    sTemp := 'IF(state,1,0))';

    StrConcatA(
        ADR(sTemp),
        ADR(sSQL),
        TO_INT(SIZEOF(sSQL))
    );


    // =================================================
    // WHERE
    // =================================================

    sTemp := ' FROM logs WHERE id BETWEEN ';

    StrConcatA(
        ADR(sTemp),
        ADR(sSQL),
        TO_INT(SIZEOF(sSQL))
    );

    sTemp := DWORD_TO_STRING(dwStartId);

    StrConcatA(
        ADR(sTemp),
        ADR(sSQL),
        TO_INT(SIZEOF(sSQL))
    );

    sTemp := ' AND ';

    StrConcatA(
        ADR(sTemp),
        ADR(sSQL),
        TO_INT(SIZEOF(sSQL))
    );


	sTemp := UDINT_TO_STRING(TO_UDINT(dwStartId) + TO_UDINT(uiCount));
	 
    StrConcatA(
        ADR(sTemp),
        ADR(sSQL),
        TO_INT(SIZEOF(sSQL))
    );

    // =================================================
    // ORDER
    // =================================================

    sTemp := ' ORDER BY id DESC;';

    StrConcatA(
        ADR(sTemp),
        ADR(sSQL),
        TO_INT(SIZEOF(sSQL))
    );

   

    // =================================================
    // MARIADB COMMAND
    // =================================================

    sCommand := '';

    sTemp :=
        'mariadb --socket=/var/lib/mysql/mysql.sock ';

    StrConcatA(
        ADR(sTemp),
        ADR(sCommand),
        TO_INT(SIZEOF(sCommand))
    );


    sTemp :=
        '-u root -pCTA-MariaDb1981! ';

    StrConcatA(
        ADR(sTemp),
        ADR(sCommand),
        TO_INT(SIZEOF(sCommand))
    );


    sTemp :=
        '--default-character-set=utf8mb4 CtaMariaDb ';

    StrConcatA(
        ADR(sTemp),
        ADR(sCommand),
        TO_INT(SIZEOF(sCommand))
    );


    sTemp :=
        '-N -B -e "';

    StrConcatA(
        ADR(sTemp),
        ADR(sCommand),
        TO_INT(SIZEOF(sCommand))
    );


    // SQL anhängen

    StrConcatA(
        ADR(sSQL),
        ADR(sCommand),
        TO_INT(SIZEOF(sCommand))
    );


    sTemp := '"';

    StrConcatA(
        ADR(sTemp),
        ADR(sCommand),
        TO_INT(SIZEOF(sCommand))
    );


    // =================================================
    // SQL AUSFÜHREN
    // =================================================

    sStdOut := '';

    diStdOutLen :=
        SysProcess_Implementation.SysProcessExecuteCommand2(
            pszCommand := sCommand,
            pszStdOut := sStdOut,
            udiStdOutLen := SIZEOF(sStdOut),
            pResult := ADR(Result)
        );


    // =================================================
    // FEHLER
    // =================================================

    IF Result <> CmpErrors.Errors.ERR_OK THEN

        xError := TRUE;
        xDone := FALSE;
        dwResult := 2;

    ELSE

        // =============================================
        // ERGEBNIS PARSEN
        // =============================================

        sRemaining := sStdOut;

        uiRead := 0;


        FOR i := 0 TO 13 DO

            IF uiRead >= uiCount THEN
                EXIT;
            END_IF;


            // -----------------------------------------
            // nächste Zeile suchen
            // MARIADB -B liefert LF
            // -----------------------------------------

            iPos := StrFindA(ADR(sRemaining), ADR(cLF),0);


            IF iPos > 0 THEN

                StrMidA(ADR(sRemaining),SIZEOF(sRemaining),iPos - 1,1,ADR(sRow),SIZEOF(sRow));

                StrDeleteA(ADR(sRemaining),  iPos,1);

            ELSE

                // letzte Zeile

                sRow := sRemaining;
                sRemaining := '';

            END_IF;


            // -----------------------------------------
            // leere Zeile ignorieren
            // -----------------------------------------

            IF LEN(sRow) > 0 THEN


                // =====================================
                // FELD 1 - ID
                // =====================================

                iPos := FIND(sRow, '\t');

                IF iPos > 0 THEN

                    sField := LEFT(sRow, iPos - 1);

                    StrDeleteA(ADR(sRow),iPos + 1,1);

                    aLogs[uiRead].id := TO_ULINT(sField);

                END_IF;


                // =====================================
                // FELD 2 - CREATED AT
                // =====================================

                iPos := FIND(sRow, '\t');

                IF iPos > 0 THEN

                    sField := LEFT(sRow, iPos - 1);

					StrDeleteA(ADR(sRow),iPos + 1,1);

                    IF LEN(sField) > 0 THEN
						sField := REPLACE(sField,'-',1,FIND(sField,' '));
                        aLogs[uiRead].createdAt := TO_DT(CONCAT('DT#',sField));
                    END_IF;

                END_IF;


                // =====================================
                // FELD 3 - EVENT TYPE
                // =====================================

                iPos := FIND(sRow, '\t');

                IF iPos > 0 THEN

                    sField := LEFT(sRow, iPos - 1);

					StrDeleteA(ADR(sRow),iPos + 1,1);

                    IF sField = 'ERROR' THEN
                        aLogs[uiRead].reportType :=
                            enReportType.Error;

                    ELSIF sField = 'WARNING' THEN
                        aLogs[uiRead].reportType :=
                            enReportType.Warning;

                    ELSIF sField = 'INFO' THEN
                        aLogs[uiRead].reportType :=
                            enReportType.Info;

                    ELSE
                        aLogs[uiRead].reportType :=
                            enReportType.Info;
                    END_IF;

                END_IF;


                // =====================================
                // FELD 4 - EVENT ID
                // =====================================

                iPos := FIND(sRow, '\t');

                IF iPos > 0 THEN

                    sField := LEFT(sRow, iPos - 1);

					StrDeleteA(ADR(sRow),iPos + 1,1);

                    aLogs[uiRead].reportId :=
                        TO_ULINT(sField);

                END_IF;


                // =====================================
                // FELD 5 - OBJECT NAME
                // =====================================

                iPos := FIND(sRow, '\t');

                IF iPos > 0 THEN

                    aLogs[uiRead].reporterText :=
                        LEFT(sRow, iPos - 1);

					StrDeleteA(ADR(sRow),iPos + 1,1);

                END_IF;


                // =====================================
                // FELD 6 - REPORT TEXT
                // =====================================

                iPos := FIND(sRow, '\t');

                IF iPos > 0 THEN

                    aLogs[uiRead].reportText :=
                        LEFT(sRow, iPos - 1);

					StrDeleteA(ADR(sRow),iPos + 1,1);

                END_IF;


                // =====================================
                // FELD 7 - DT FROM
                // =====================================

                iPos := FIND(sRow, '\t');

                IF iPos > 0 THEN

                    sField := LEFT(sRow, iPos - 1);

					StrDeleteA(ADR(sRow),iPos + 1,1);

                    IF LEN(sField) > 0 THEN
						sField := REPLACE(sField,'-',1,FIND(sField,' '));
                        aLogs[uiRead].dtFrom := TO_DT(CONCAT('DT#',sField));
                    END_IF;

                END_IF;


                // =====================================
                // FELD 8 - DT TO
                // =====================================

                iPos := FIND(sRow, '\t');

                IF iPos > 0 THEN

                    sField := LEFT(sRow, iPos - 1);

					StrDeleteA(ADR(sRow),iPos + 1,1);

                    IF LEN(sField) > 0 THEN
						sField := REPLACE(sField,'-',1,FIND(sField,' '));
                        aLogs[uiRead].dtTo := TO_DT(CONCAT('DT#',sField));
                    END_IF;

                END_IF;


                // =====================================
                // FELD 9 - IS QUITT
                // =====================================

                iPos := FIND(sRow, '\t');

                IF iPos > 0 THEN

                    sField := LEFT(sRow, iPos - 1);

					StrDeleteA(ADR(sRow),iPos + 1,1);

                    aLogs[uiRead].isQuitt := TO_BOOL(TO_INT(sField));

                END_IF;


                // =====================================
                // FELD 10 - REPORT TEXT LIST
                // =====================================

                iPos := FIND(sRow, '\t');

                IF iPos > 0 THEN

                    aLogs[uiRead].reportTextList :=
                        LEFT(sRow, iPos - 1);

					StrDeleteA(ADR(sRow),iPos + 1,1);

                END_IF;


                // =====================================
                // FELD 11 - TEXT ID
                // =====================================

                iPos := FIND(sRow, '\t');

                IF iPos > 0 THEN

                    sField := LEFT(sRow, iPos - 1);

					StrDeleteA(ADR(sRow),iPos + 1,1);

                    aLogs[uiRead].reportTextId :=
                        sField;

                END_IF;


                // =====================================
                // FELD 12 - ACKNOWLEDGEMENT
                // =====================================

                iPos := FIND(sRow, '\t');

                IF iPos > 0 THEN

                    sField := LEFT(sRow, iPos - 1);

					StrDeleteA(ADR(sRow),iPos + 1,1);

                    aLogs[uiRead].reportAcknowledgType :=
                        TO_USINT(sField);

                END_IF;


                // =====================================
                // FELD 13 - OBJECT ID
                // =====================================

                iPos := FIND(sRow, '\t');

                IF iPos > 0 THEN

                    aLogs[uiRead].objectId :=
                        LEFT(sRow, iPos - 1);

					StrDeleteA(ADR(sRow),iPos + 1,1);

                END_IF;


                // =====================================
                // FELD 14 - INSTANCE PATH
                // =====================================

                iPos := FIND(sRow, '\t');

                IF iPos > 0 THEN

                    aLogs[uiRead].instancePath :=
                        LEFT(sRow, iPos - 1);

					StrDeleteA(ADR(sRow),iPos + 1,1);

                END_IF;


                // =====================================
                // FELD 15 - ADDITIONAL TEXT
                // =====================================

                iPos := FIND(sRow, '\t');

                IF iPos > 0 THEN

                    aLogs[uiRead].additionalText :=
                        LEFT(sRow, iPos - 1);

					StrDeleteA(ADR(sRow),iPos + 1,1);

                END_IF;


                // =====================================
                // FELD 16 - PRIO
                // =====================================

                iPos := FIND(sRow, '\t');

                IF iPos > 0 THEN

                    sField := LEFT(sRow, iPos - 1);

					StrDeleteA(ADR(sRow),iPos + 1,1);

                    aLogs[uiRead].prio :=
                        TO_USINT(sField);

                END_IF;


                // =====================================
                // FELD 17 - IN STATE
                // =====================================

                iPos := FIND(sRow, '\t');

                IF iPos > 0 THEN

                    sField := LEFT(sRow, iPos - 1);

					StrDeleteA(ADR(sRow),iPos + 1,1);

                    aLogs[uiRead].reportIn := TO_BOOL(TO_INT(sField));
                END_IF;


                // =====================================
                // FELD 18 - STATE
                // =====================================

                IF LEN(sRow) > 0 THEN

                    aLogs[uiRead].stateActive := TO_BOOL(TO_INT(sRow));

                END_IF;


                // =====================================
                // DATENSATZ GÜLTIG
                // =====================================

                IF aLogs[uiRead].id > 0 THEN

                    uiRead := uiRead + 1;

                END_IF;

            END_IF;

        END_FOR;


        // =============================================
        // ERGEBNIS
        // =============================================

        uiCountRead := uiRead;

        IF uiRead > 0 THEN

            xDone := TRUE;
            xError := FALSE;
            dwResult := 0;

        ELSE

            xDone := TRUE;
            xError := FALSE;
            dwResult := 0;

        END_IF;

    END_IF;

END_IF;


// =====================================================
// BUSY
// =====================================================

IF xExecute AND NOT xExecuteOld THEN
    xBusy := TRUE;
ELSE
    xBusy := FALSE;
END_IF;


// =====================================================
// FLANKE SPEICHERN
// =====================================================

xExecuteOld := xExecute;

END_FUNCTION

// 30 Program Organization Units/SORT/fbSort
FUNCTION_BLOCK fbSort
VAR_INPUT
END_VAR
VAR_OUTPUT
END_VAR
VAR
    uiAnzAktivError             :   UINT;
    uiAnzAktivWarning           :   UINT;
    uiAnzAktivInfo              :   UINT;
    uiAnzAktivReports           :   UINT;
    uiAnzAktivReportsInTable    :   UINT;
END_VAR

METHOD metSortPrio : BOOL
VAR_INPUT
END_VAR
VAR
    diFor1    : DINT;
    diFor2    : DINT;
    itfTempt  : ITF_REPORTOBJECT;
    diCounts  : DINT;
END_VAR
(* Reset *)
FOR diFor1 := 1 TO Parameter.diMaxObject DO
		GVL_Report.ayItfAktiveReports[diFor1] := 0;
END_FOR;
uiAnzAktivError             := 0;
uiAnzAktivWarning           := 0;
uiAnzAktivInfo              := 0;
uiAnzAktivReports           := 0;

(* Get Aktive Reports *)
FOR diFor1 := 1 TO Parameter.diMaxObject DO
	IF GVL_Report.ayReportObject[diFor1].proStateActive THEN
		diCounts := LIMIT(1,diCounts + 1, Parameter.diMaxObject);
		GVL_Report.ayItfAktiveReports[diCounts] := GVL_Report.ayReportObject[diFor1];
		IF GVL_Report.ayItfAktiveReports[diCounts].proReportType = enReportType.Error THEN
			uiAnzAktivError     := uiAnzAktivError + 1;
		ELSIF GVL_Report.ayItfAktiveReports[diCounts].proReportType = enReportType.Warning THEN
			uiAnzAktivWarning   := uiAnzAktivWarning + 1;
		ELSIF GVL_Report.ayItfAktiveReports[diCounts].proReportType = enReportType.Info THEN
			uiAnzAktivInfo      := uiAnzAktivInfo + 1;
		END_IF
		uiAnzAktivReports := uiAnzAktivError + uiAnzAktivWarning + uiAnzAktivInfo;
	END_IF;
END_FOR;

(* Sort Aktive Reports dt *)
FOR diFor1 := 1 TO diCounts DO
	FOR diFor2 := 1 TO diCounts -1 DO
		(* Sort nach Typ *)
		IF GVL_Report.ayItfAktiveReports[diFor2].proDtFrom < GVL_Report.ayItfAktiveReports[diFor2 + 1].proDtFrom THEN
			itfTempt                                    := GVL_Report.ayItfAktiveReports[diFor2]; 
			GVL_Report.ayItfAktiveReports[diFor2]       := GVL_Report.ayItfAktiveReports[diFor2 + 1];
			GVL_Report.ayItfAktiveReports[diFor2 + 1]   := itfTempt;         
		END_IF;     
	END_FOR;
END_FOR

GVL_Report.ayItfSortetReportsPrio := GVL_Report.ayItfAktiveReports;
(* Sort *)
FOR diFor1 := 1 TO diCounts DO
	FOR diFor2 := 1 TO diCounts -1 DO
		(* Sort nach Typ *)
		IF __QUERYINTERFACE(GVL_Report.ayItfSortetReportsPrio[diFor2],GVL_Report.ayItfSortetReportsPrio[diFor2]) AND __QUERYINTERFACE(GVL_Report.ayItfSortetReportsPrio[diFor2 + 1],GVL_Report.ayItfSortetReportsPrio[diFor2 + 1]) THEN
			IF GVL_Report.ayItfSortetReportsPrio[diFor2].proReportType < GVL_Report.ayItfSortetReportsPrio[diFor2 + 1].proReportType THEN
				itfTempt                                        := GVL_Report.ayItfSortetReportsPrio[diFor2]; 
				GVL_Report.ayItfSortetReportsPrio[diFor2]       := GVL_Report.ayItfSortetReportsPrio[diFor2 + 1];
				GVL_Report.ayItfSortetReportsPrio[diFor2 + 1]   := itfTempt; 
			(* Sort nach Prio wenn Typ gleich *)    
			ELSIF GVL_Report.ayItfSortetReportsPrio[diFor2].proReportType = GVL_Report.ayItfSortetReportsPrio[diFor2 + 1].proReportType THEN
				IF GVL_Report.ayItfSortetReportsPrio[diFor2].proPrio > GVL_Report.ayItfSortetReportsPrio[diFor2 + 1].proPrio AND GVL_Report.ayItfSortetReportsPrio[diFor2 + 1].proPrio >= 1 THEN
					itfTempt                                        := GVL_Report.ayItfSortetReportsPrio[diFor2]; 
					GVL_Report.ayItfSortetReportsPrio[diFor2]       := GVL_Report.ayItfSortetReportsPrio[diFor2 + 1];
					GVL_Report.ayItfSortetReportsPrio[diFor2 + 1]   := itfTempt;                
				END_IF;           
			END_IF;     
		END_IF;
	END_FOR;
END_FOR;
GVL_Report.fbReportVisu.metReload();
END_METHOD

METHOD metFilterCustom : BOOL
VAR_INPUT
    usiFilter   :   USINT;
	diClientId	:	DINT;
END_VAR
VAR
    diFor1          : DINT;
    diFor2          : DINT;
    itfTempt        : ITF_REPORTOBJECT;
    diCounts        : DINT;
    diCountsFilter  : DINT;
    usiSort         : USINT;
END_VAR
FOR diFor1 := 1 TO Parameter.diMaxObject DO
        GVL_Report.ayItfSortetReportsCustom[diClientId][diFor1] := 0;
END_FOR;
(* Filter *)
CASE usiFilter OF
    0:(* No Filter *)
        FOR diFor1 := 1 TO Parameter.diMaxObject DO
            IF GVL_Report.ayItfSortetReportsPrio[diFor1] <> 0 THEN
                IF GVL_Report.ayItfSortetReportsPrio[diFor1].proStateActive THEN
                    diCounts := LIMIT(1,diCounts + 1, Parameter.diMaxObject);
                    GVL_Report.ayItfSortetReportsCustom[diClientId][diCounts] := GVL_Report.ayItfSortetReportsPrio[diFor1];
                END_IF;
            END_IF;
        END_FOR;   
        uiAnzAktivReportsInTable := uiAnzAktivReports;
    1:(* Only Error *)
        FOR diFor1 := 1 TO Parameter.diMaxObject DO
            IF GVL_Report.ayItfSortetReportsPrio[diFor1] <> 0 THEN
                IF GVL_Report.ayItfSortetReportsPrio[diFor1].proStateActive AND_THEN GVL_Report.ayItfSortetReportsPrio[diFor1].proReportType = enReportType.Error THEN
                    diCounts := LIMIT(1,diCounts + 1, Parameter.diMaxObject);
                    GVL_Report.ayItfSortetReportsCustom[diClientId][diCounts] := GVL_Report.ayItfSortetReportsPrio[diFor1];
                END_IF;
            END_IF;
        END_FOR;    
        uiAnzAktivReportsInTable := uiAnzAktivError;
    2:(* Only Warning *)
        FOR diFor1 := 1 TO Parameter.diMaxObject DO
            IF GVL_Report.ayItfSortetReportsPrio[diFor1] <> 0 THEN
                IF GVL_Report.ayItfSortetReportsPrio[diFor1].proStateActive AND_THEN GVL_Report.ayItfSortetReportsPrio[diFor1].proReportType = enReportType.Warning THEN
                    diCounts := LIMIT(1,diCounts + 1, Parameter.diMaxObject);
                    GVL_Report.ayItfSortetReportsCustom[diClientId][diCounts] := GVL_Report.ayItfSortetReportsPrio[diFor1];
                END_IF;
            END_IF;
        END_FOR;      
        uiAnzAktivReportsInTable := uiAnzAktivWarning;
    3:(* Only Info *)
        FOR diFor1 := 1 TO Parameter.diMaxObject DO
            IF GVL_Report.ayItfSortetReportsPrio[diFor1] <> 0 THEN
                IF GVL_Report.ayItfSortetReportsPrio[diFor1].proStateActive AND_THEN GVL_Report.ayItfSortetReportsPrio[diFor1].proReportType = enReportType.Info THEN
                    diCounts := LIMIT(1,diCounts + 1, Parameter.diMaxObject);
                    GVL_Report.ayItfSortetReportsCustom[diClientId][diCounts] := GVL_Report.ayItfSortetReportsPrio[diFor1];
                END_IF;
            END_IF;
        END_FOR;    
        uiAnzAktivReportsInTable := uiAnzAktivInfo;    
    4:(* Error and Warning *)
        FOR diFor1 := 1 TO Parameter.diMaxObject DO
            IF GVL_Report.ayItfSortetReportsPrio[diFor1] <> 0 THEN
                IF GVL_Report.ayItfSortetReportsPrio[diFor1].proStateActive AND_THEN 
                   GVL_Report.ayItfSortetReportsPrio[diFor1].proReportType = enReportType.Error OR GVL_Report.ayItfSortetReportsPrio[diFor1].proReportType = enReportType.Warning THEN
                    diCounts := LIMIT(1,diCounts + 1, Parameter.diMaxObject);
                    GVL_Report.ayItfSortetReportsCustom[diClientId][diCounts] := GVL_Report.ayItfSortetReportsPrio[diFor1];
                END_IF;
            END_IF;
        END_FOR;       
        uiAnzAktivReportsInTable := uiAnzAktivError + uiAnzAktivWarning;
    5:(* Error and Info *)
        FOR diFor1 := 1 TO Parameter.diMaxObject DO
            IF GVL_Report.ayItfSortetReportsPrio[diFor1] <> 0 THEN
                IF GVL_Report.ayItfSortetReportsPrio[diFor1].proStateActive AND_THEN 
                   GVL_Report.ayItfSortetReportsPrio[diFor1].proReportType = enReportType.Error OR GVL_Report.ayItfSortetReportsPrio[diFor1].proReportType = enReportType.Info THEN
                    diCounts := LIMIT(1,diCounts + 1, Parameter.diMaxObject);
                    GVL_Report.ayItfSortetReportsCustom[diClientId][diCounts] := GVL_Report.ayItfSortetReportsPrio[diFor1];
                END_IF;
            END_IF;
        END_FOR;           
        uiAnzAktivReportsInTable := uiAnzAktivError + uiAnzAktivInfo;
    6:(* Warning and Info *)
        FOR diFor1 := 1 TO Parameter.diMaxObject DO
            IF GVL_Report.ayItfSortetReportsPrio[diFor1] <> 0 THEN
                IF GVL_Report.ayItfSortetReportsPrio[diFor1].proStateActive AND_THEN 
                   GVL_Report.ayItfSortetReportsPrio[diFor1].proReportType = enReportType.Warning OR GVL_Report.ayItfSortetReportsPrio[diFor1].proReportType = enReportType.Info THEN
                    diCounts := LIMIT(1,diCounts + 1, Parameter.diMaxObject);
                    GVL_Report.ayItfSortetReportsCustom[diClientId][diCounts] := GVL_Report.ayItfSortetReportsPrio[diFor1];
                END_IF;
            END_IF;
        END_FOR;        
        uiAnzAktivReportsInTable := uiAnzAktivWarning + uiAnzAktivInfo;
    ELSE
        usiFilter := 0;     
END_CASE


(* Sort *)
CASE usiSort OF
    0:(* Sort Type and Prio *) 
        FOR diFor1 := 1 TO diCounts DO
            FOR diFor2 := 1 TO diCounts -1 DO
                (* Sort nach Typ *)
                IF GVL_Report.ayItfSortetReportsCustom[diClientId][diFor2].proReportType < GVL_Report.ayItfSortetReportsCustom[diClientId][diFor2 + 1].proReportType THEN
                    itfTempt                                            := GVL_Report.ayItfSortetReportsCustom[diClientId][diFor2]; 
                    GVL_Report.ayItfSortetReportsCustom[diClientId][diFor2]         := GVL_Report.ayItfSortetReportsCustom[diClientId][diFor2 + 1];
                    GVL_Report.ayItfSortetReportsCustom[diClientId][diFor2 + 1]     := itfTempt; 
                (* Sort nach Prio wenn Typ gleich *)    
                ELSIF GVL_Report.ayItfSortetReportsCustom[diClientId][diFor2].proReportType = GVL_Report.ayItfSortetReportsCustom[diClientId][diFor2 + 1].proReportType THEN
                    IF GVL_Report.ayItfSortetReportsCustom[diClientId][diFor2].proPrio > GVL_Report.ayItfSortetReportsCustom[diClientId][diFor2 + 1].proPrio AND GVL_Report.ayItfSortetReportsCustom[diClientId][diFor2 + 1].proPrio >= 1 THEN
                        itfTempt                                        := GVL_Report.ayItfSortetReportsCustom[diClientId][diFor2]; 
                        GVL_Report.ayItfSortetReportsCustom[diClientId][diFor2]     := GVL_Report.ayItfSortetReportsCustom[diClientId][diFor2 + 1];
                        GVL_Report.ayItfSortetReportsCustom[diClientId][diFor2 + 1] := itfTempt;                
                    END_IF           
                END_IF;     
            END_FOR;
        END_FOR;  
    ELSE
        usiSort := 0;
END_CASE
END_METHOD

PROPERTY proAnzAktiveError : UINT
GET
proAnzAktiveError := uiAnzAktivError;
END_GET
END_PROPERTY

PROPERTY proAnzAktiveInfo : UINT
GET
proAnzAktiveInfo := uiAnzAktivInfo;
END_GET
END_PROPERTY

PROPERTY proAnzAktiveReports : UINT
GET
proAnzAktiveReports := uiAnzAktivReports;
END_GET
END_PROPERTY

PROPERTY proAnzAktiveWarning : UINT
GET
proAnzAktiveWarning:= uiAnzAktivWarning;
END_GET
END_PROPERTY

PROPERTY proAnzReportsInTable : UINT
GET
proAnzReportsInTable := uiAnzAktivReportsInTable;
END_GET
END_PROPERTY

END_FUNCTION_BLOCK

// 30 Program Organization Units/SQL/Fc_MariaDbDeleteHistory
FUNCTION Fc_MariaDbDeleteHistory
VAR_INPUT
    xExecute 			   : BOOL;
END_VAR

VAR_OUTPUT
    xBusy       : BOOL;
    xDone       : BOOL;
    xError      : BOOL;
    dwResult    : DWORD;
END_VAR

VAR
    sCommand    : STRING(1024);
    sStdOut     : STRING(100);	
	sFind		: STRING := 'MAX(id)$N';
    xExecuteOld : BOOL;

	sTemp		: STRING(1024);
    Result      : RTS_IEC_RESULT;

    diStdOutLen : DINT;
END_VAR

// Ausgänge zurücksetzen
xDone := FALSE;
xError := FALSE;
xBusy := TRUE;
dwResult := 0;
sStdOut := '';
sTemp	:= '';
sCommand:= '';

// =====================================================
// LINUX COMMAND
// =====================================================
sCommand := '';
sTemp := '';
sTemp := 'mariadb --socket=/var/lib/mysql/mysql.sock -u root -pCTA-MariaDb1981! --default-character-set=utf8mb4 CtaMariaDb -e "TRUNCATE TABLE logs;"';
StrConcatA(ADR(sTemp),ADR(sCommand),TO_INT(SIZEOF(sCommand)));

// =====================================================
// SYSPROCESS
// =====================================================

diStdOutLen :=
	SysProcess_Implementation.SysProcessExecuteCommand2(
		pszCommand := sCommand,
		pszStdOut := sStdOut,
		udiStdOutLen := SIZEOF(sStdOut),
		pResult := ADR(Result)
	);

// =====================================================
// ERGEBNIS
// =====================================================

IF Result = CmpErrors.Errors.ERR_OK THEN

	xDone := TRUE;
	xError := FALSE;

ELSE

	xDone := FALSE;
	xError := TRUE;

END_IF;

xBusy := FALSE;

END_FUNCTION

// 30 Program Organization Units/OBJ/fcReportIdToString8
FUNCTION fcReportIdToString8 : STRING(10)
VAR_INPUT
    uliReportId :   ULINT;
END_VAR
VAR
END_VAR

fcReportIdToString8 := '          ';
IF uliReportId > 0 THEN 
    fcReportIdToString8 := REPLACE(fcReportIdToString8,TO_STRING(uliReportId),LEN(TO_STRING(uliReportId)),1); 
END_IF;

END_FUNCTION

// 30 Program Organization Units/OBJ/fbReportObject
{attribute 'enable_dynamic_creation'}
FUNCTION_BLOCK fbReportObject EXTENDS CtaAppBmk.fbBMK IMPLEMENTS ITF_REPORTOBJECT
VAR
    scReportMetaData    		: scReportMetaData;
	fbLogString					: CtaAppInfluxLog.FB_LOG_NODE_STRING;
    xSaveOnChange       		: BOOL;
    xFirstTryTextLoad   		: BOOL;
	xFirstTryTextLoadLanguage   : BOOL;
    TON_GARBAGE        			: TON;
    xGarbageControll    		: BOOL;
END_VAR

PROPERTY FINAL proGetReporterText : STRING[150]
GET
IF proGetVendorDesignation <> '' AND proGetBMK <> '' THEN
    proGetReporterText := CONCAT(proGetBMK,CONCAT(' ',proGetVendorDesignation));
ELSE
    proGetReporterText := proGetInstancePath;
END_IF;
END_GET
END_PROPERTY

PROPERTY FINAL proGetReportText : STRING[140]
GET
VAR
    stTempText  	:   STRING[140];
    dwState     	:   DWORD;
	ITextListInfo	:	TLU.ITextListInfo;
END_VAR
stTempText := '';
(*Load Text By Language*)
	ITextListInfo := TLU.GetTextListInfo(scReportMetaData.stReportTextList);
	IF __QUERYINTERFACE(ITextListInfo,ITextListInfo) THEN
		dwState := TLU.GetText(scReportMetaData.stReportTextList,scReportMetaData.stReportTxtId,ADR(stTempText),SIZEOF(stTempText)-SIZEOF(scReportMetaData.stAdditionalText));
		IF stTempText = '' AND NOT xFirstTryTextLoad THEN
			dwState := TLU.GetText(scReportMetaData.stReportTextList,scReportMetaData.stReportTxtId,ADR(stTempText),SIZEOF(stTempText)-SIZEOF(scReportMetaData.stAdditionalText));
			xFirstTryTextLoad := TRUE;
		END_IF; 
		(* Concat Additional Text to Repor*)
		IF scReportMetaData.stAdditionalText <> '' THEN
			stTempText := CONCAT(stTempText,CONCAT(' ',scReportMetaData.stAdditionalText));
		END_IF;
		ITextListInfo.Release();
	ELSE
		scReportMetaData.stReportTextList :='CtaAppReport.txtNoTextList';
		scReportMetaData.stReportTxtId 	  := '1';
		dwState := TLU.GetText(scReportMetaData.stReportTextList,scReportMetaData.stReportTxtId,ADR(stTempText),SIZEOF(stTempText)-SIZEOF(scReportMetaData.stAdditionalText));
		IF stTempText = '' AND NOT xFirstTryTextLoad THEN
			dwState := TLU.GetText(scReportMetaData.stReportTextList,scReportMetaData.stReportTxtId,ADR(stTempText),SIZEOF(stTempText)-SIZEOF(scReportMetaData.stAdditionalText));
			xFirstTryTextLoad := TRUE;
		END_IF; 
		(* Concat Additional Text to Repor*)
		IF scReportMetaData.stAdditionalText <> '' THEN
			stTempText := CONCAT(stTempText,CONCAT(' ',scReportMetaData.stAdditionalText));
		END_IF;		
	END_IF;
    (* Write Text to Output*)
    proGetReportText := stTempText;
END_GET
END_PROPERTY

PROPERTY FINAL proAdditionalText : STRING(20)
GET
proAdditionalText := scReportMetaData.stAdditionalText;
END_GET
SET
IF scReportMetaData.stAdditionalText <> proAdditionalText THEN
    scReportMetaData.stAdditionalText := proAdditionalText;
END_IF;
END_SET
END_PROPERTY

PROPERTY FINAL proCountRetry : INT
GET
proCountRetry := scReportMetaData.iCountRetry;
END_GET
SET
IF scReportMetaData.iCountRetry <> proCountRetry THEN    
    scReportMetaData.iCountRetry := proCountRetry;
END_IF;
END_SET
END_PROPERTY

PROPERTY FINAL proIsQuitt : BOOL
GET
proIsQuitt := scReportMetaData.xIsQuitt;
END_GET
SET
IF scReportMetaData.xIsQuitt <> proIsQuitt THEN
    scReportMetaData.xIsQuitt := proIsQuitt;
    xSaveOnChange := TRUE;
END_IF;
END_SET
END_PROPERTY

PROPERTY FINAL proIsSelected : BOOL
GET
proIsSelected := scReportMetaData.xIsSelected;
END_GET
SET
IF scReportMetaData.xIsSelected <> proIsSelected THEN
    scReportMetaData.xIsSelected := proIsSelected;
END_IF;
END_SET
END_PROPERTY

PROPERTY FINAL proMaxRetry : INT
GET
proMaxRetry := scReportMetaData.iMaxRetry;
END_GET
SET
IF scReportMetaData.iMaxRetry <> proMaxRetry THEN
    scReportMetaData.iMaxRetry := proMaxRetry;
END_IF;
END_SET
END_PROPERTY

PROPERTY FINAL proReportAcknowledgType : enReportacknowledgeType
GET
proReportAcknowledgType := scReportMetaData.enReportacknowledgeType;
END_GET
SET
IF scReportMetaData.enReportacknowledgeType <> proReportAcknowledgType THEN
    scReportMetaData.enReportacknowledgeType := proReportAcknowledgType;
END_IF;
END_SET
END_PROPERTY

PROPERTY FINAL proReportId : ULINT
GET
proReportId := scReportMetaData.uliReportId;
END_GET
END_PROPERTY

PROPERTY FINAL proReportTextId : STRING(3)
GET
proReportTextId := scReportMetaData.stReportTxtId;
END_GET
SET
IF scReportMetaData.stReportTxtId <> proReportTextId THEN
    scReportMetaData.stReportTxtId := proReportTextId;
END_IF;
END_SET
END_PROPERTY

PROPERTY FINAL proReportTextList : STRING(100)
GET
proReportTextList := scReportMetaData.stReportTextList;
END_GET
SET
IF scReportMetaData.stReportTextList <> proReportTextList THEN
    scReportMetaData.stReportTextList := proReportTextList;
END_IF;
END_SET
END_PROPERTY

PROPERTY FINAL proReportType : enReportType
GET
proReportType := scReportMetaData.enReportType;
END_GET
SET
IF proReportType <> scReportMetaData.enReportType THEN
    scReportMetaData.enReportType := proReportType;
END_IF;
END_SET
END_PROPERTY

PROPERTY FINAL proReporterObjectId : STRING(20)
GET
proReporterObjectId := scReportMetaData.stReporterObjId;
END_GET
SET
IF scReportMetaData.stReporterObjId <> proReporterObjectId THEN
    scReportMetaData.stReporterObjId := proReporterObjectId;
    stObjId := proReporterObjectId;
END_IF;
END_SET
END_PROPERTY

PROPERTY FINAL proStateActive : BOOL
GET
proStateActive := scReportMetaData.xActive;
END_GET
SET
IF scReportMetaData.xActive <> proStateActive THEN
    scReportMetaData.xActive := proStateActive;
    xSaveOnChange := TRUE;
END_IF;
END_SET
END_PROPERTY

PROPERTY FINAL proWritePosInCsv : DWORD
GET
proWritePosInCsv := scReportMetaData.dwWritePosInCsv;
END_GET
SET
scReportMetaData.dwWritePosInCsv := proWritePosInCsv;
END_SET
END_PROPERTY

PROPERTY FINAL proQuitt : BOOL
SET
IF proQuitt <> scReportMetaData.xQuitt THEN
    scReportMetaData.xQuitt := proQuitt;
    IF proQuitt THEN
        proIsQuitt              := TRUE;
    END_IF;
END_IF;
END_SET
GET
proQuitt := scReportMetaData.xQuitt;
END_GET
END_PROPERTY

METHOD PRIVATE FINAL metSendDataToInflux : BOOL
(* Enable Log *)
fbLogString.ENABLE 			:= TRUE;
(* Check BMK *)
IF NOT proNoBmkInList THEN
	fbLogString.SET_VALUE := CONCAT(proGetBMK,CONCAT(' ',proGetReportText));
ELSE
	IF FIND(proGetReporterText,'Steuerung.Application.') > 0 THEN
		fbLogString.SET_VALUE := CONCAT(DELETE(proGetReporterText,LEN('Steuerung.Application.'),FIND(proGetReporterText,'Steuerung.Application.')),CONCAT(' ',proGetReportText)); 
	ELSE
		fbLogString.SET_VALUE := CONCAT(proGetReporterText,CONCAT(' ',proGetReportText));
	END_IF;
END_IF;
   
(* Report Type *)
IF scReportMetaData.enReportType = enReportType.Error THEN
    fbLogString.KEY   := 'Error';
ELSIF scReportMetaData.enReportType = enReportType.Warning THEN
    fbLogString.KEY   := 'Warning';
ELSIF scReportMetaData.enReportType = enReportType.Info THEN
    fbLogString.KEY   := 'Info';
END_IF;
(* Destroy after Send *)
fbLogString.DESTROYAFTERLOG := TRUE;
END_METHOD

METHOD FINAL metReportObject : BOOL
VAR_INPUT
END_VAR
(* Type of Acknowledge *)
IF scReportMetaData.enReportacknowledgeType = enReportacknowledgeType.Auto AND NOT scReportMetaData.xIsQuitt THEN
    scReportMetaData.xIsQuitt   := TRUE;
ELSIF scReportMetaData.enReportacknowledgeType = enReportacknowledgeType.RetryN THEN 
    IF scReportMetaData.iCountRetry < scReportMetaData.iMaxRetry AND NOT scReportMetaData.xIsQuitt THEN
        scReportMetaData.enReportacknowledgeType    := enReportacknowledgeType.Auto;
        scReportMetaData.xIsQuitt                   := TRUE;
    ELSE
        scReportMetaData.enReportacknowledgeType    := enReportacknowledgeType.Quit;
    END_IF;    
END_IF;
IF scReportMetaData.xReportIn THEN
    IF NOT scReportMetaData.xActive THEN       
        // Set State Active 
        scReportMetaData.xActive := TRUE;
        // Set Dt From
        scReportMetaData.dtFrom := CtaAppTime.FuGetLocalDateAndTime();
        // Set Id
        IF scReportMetaData.uliReportId = 0 THEN
            scReportMetaData.uliReportId := fcBmkToId(proGetBMK,TO_DINT(scReportMetaData.stReportTxtId),FALSE,scReportMetaData.enReportType);
        END_IF  
        // Write Dt From To Csv
        metWriteDtFromToCsv();
        GVL_Report.fbSort.metSortPrio();     
        metSendDataToInflux();
        IF scReportMetaData.enReportType = enReportType.Error THEN
            GVL_REPORT_PERSISTENT.scLastErrorReport    := scReportMetaData;
        ELSIF scReportMetaData.enReportType = enReportType.Warning THEN
            GVL_REPORT_PERSISTENT.scLastWarningReport  := scReportMetaData;
        ELSIF scReportMetaData.enReportType = enReportType.Info THEN
            GVL_REPORT_PERSISTENT.scLastInfoReport     := scReportMetaData;
        END_IF;    
    END_IF;
ELSE
    IF scReportMetaData.xIsQuitt AND scReportMetaData.xActive THEN    
        // Set State Inactive 
        scReportMetaData.xActive := FALSE;        
        // Write Dt To To Csv
        metWriteDtToToCsv();
        GVL_Report.fbSort.metSortPrio();  
    END_IF;    
END_IF;
metSaveOnChange();
xGarbageControll := FALSE;
END_METHOD

PROPERTY FINAL proReportIn : BOOL
SET
IF proReportIn <> scReportMetaData.xReportIn THEN
    scReportMetaData.xReportIn := proReportIn;
    xSaveOnChange := TRUE;
END_IF;
END_SET
GET
proReportIn := scReportMetaData.xReportIn;
END_GET
END_PROPERTY

PROPERTY FINAL proDtFrom : DT
SET
scReportMetaData.dtFrom := proDtFrom;
END_SET
GET
proDtFrom := scReportMetaData.dtFrom;
END_GET
END_PROPERTY

PROPERTY FINAL proDtTo : DT
SET
scReportMetaData.dtTo := proDtTo;
END_SET
GET
proDtTo := scReportMetaData.dtTo;
END_GET
END_PROPERTY

PROPERTY FINAL proSetMetaData : scReportMetaData
SET
scReportMetaData := proSetMetaData;
IF stObjId <> scReportMetaData.stReporterObjId THEN
	stObjId := scReportMetaData.stReporterObjId;
END_IF
END_SET
END_PROPERTY

METHOD FINAL metDestroy
VAR_INPUT
END_VAR
scReportMetaData.xReportIn                   := FALSE;
scReportMetaData.xActive                     := FALSE;
scReportMetaData.xIsQuitt                    := FALSE;
scReportMetaData.xQuitt                      := FALSE;
scReportMetaData.xIsSelected                 := FALSE;
scReportMetaData.dtFrom                      := DT#1970-1-1-0:0:0;
scReportMetaData.dtTo                        := DT#1970-1-1-0:0:0;
scReportMetaData.iMaxRetry                   := 0;
scReportMetaData.iCountRetry                 := 0;
scReportMetaData.stReportTxtId               := '';
scReportMetaData.stReportTextList            := '';
scReportMetaData.uliReportId                 := 0;
scReportMetaData.enReportType                := enReportType.Info;
scReportMetaData.enReportacknowledgeType     := enReportacknowledgeType.Auto;
scReportMetaData.stReporterObjId             := '';
scReportMetaData.stAdditionalText            := '';
scReportMetaData.dwWritePosInCsv             := 0;
stObjId										 := '';
proSetInstancePath						     := '';
xFirstTryTextLoad                            := FALSE;
END_METHOD

PROPERTY FINAL proPrio : USINT
SET
scReportMetaData.usiPrio := proPrio;
END_SET
GET
proPrio := scReportMetaData.usiPrio;
END_GET
END_PROPERTY

METHOD FINAL metWriteDtFromToCsv : DWORD
VAR_INPUT
END_VAR
// Write Dt From To Csv
GVL_Report.fbDataHandler.metAddObjForeWriteDtFrom(THIS^);
END_METHOD

METHOD FINAL metWriteDtToToCsv : DWORD
VAR_INPUT
END_VAR
// Set Dt To
scReportMetaData.dtTo := CtaAppTime.FuGetLocalDateAndTime();
// Write Dt To To Csv
GVL_Report.fbDataHandler.metAddObjForeWriteDtTo(THIS^);
END_METHOD

METHOD FINAL metSaveOnChange : BOOL
VAR_INPUT
END_VAR
IF xSaveOnChange THEN
    GVL_Report.fbDataHandler.metAddObjForeWriteOnChange(THIS^); 
    GVL_Report.fbReportVisu.metReload(); 
    xSaveOnChange := FALSE; 
END_IF;
END_METHOD

METHOD metGarbage : BOOL
VAR_INPUT
END_VAR
TON_GARBAGE(IN := xGarbageControll,PT := T#3S);
IF TON_GARBAGE.Q THEN
    // Set State Inactive 
    scReportMetaData.xActive := FALSE;     
    metWriteDtToToCsv();
    metDestroy();
	metGarbage := TRUE;
END_IF;
xGarbageControll := TRUE;
END_METHOD

METHOD GetReportTextLanguage : STRING[140]
VAR_INPUT
	language	:	STRING(4);
END_VAR
VAR
    stTempText  	:   STRING[140];
    dwState     	:   DWORD;
	ITextListInfo	:	TLU.ITextListInfo;
END_VAR
stTempText := '';
(*Load Text By Language*)
	ITextListInfo := TLU.GetTextListInfo(scReportMetaData.stReportTextList);
	IF __QUERYINTERFACE(ITextListInfo,ITextListInfo) THEN
		dwState := TLU.GetLanguageText(scReportMetaData.stReportTextList,scReportMetaData.stReportTxtId,language,ADR(stTempText),SIZEOF(stTempText)-SIZEOF(scReportMetaData.stAdditionalText));
		IF stTempText = '' AND NOT xFirstTryTextLoadLanguage THEN
			CmpDynamicText.DynamicTextLoadLanguage(language);
			TLU.CmpDynamicText.DynamicTextReloadTexts();
			dwState := TLU.GetLanguageText(scReportMetaData.stReportTextList,scReportMetaData.stReportTxtId,language,ADR(stTempText),SIZEOF(stTempText)-SIZEOF(scReportMetaData.stAdditionalText));
			xFirstTryTextLoadLanguage := TRUE;
		END_IF; 
		(* Concat Additional Text to Repor*)
		IF scReportMetaData.stAdditionalText <> '' THEN
			stTempText := CONCAT(stTempText,CONCAT(' ',scReportMetaData.stAdditionalText));
		END_IF;
		ITextListInfo.Release();
	ELSE
		scReportMetaData.stReportTextList :='CtaAppReport.txtNoTextList';
		scReportMetaData.stReportTxtId 	  := '1';
		dwState := TLU.GetText(scReportMetaData.stReportTextList,scReportMetaData.stReportTxtId,ADR(stTempText),SIZEOF(stTempText)-SIZEOF(scReportMetaData.stAdditionalText));
		IF stTempText = '' AND NOT xFirstTryTextLoadLanguage THEN
			CmpDynamicText.DynamicTextLoadLanguage(language);
			TLU.CmpDynamicText.DynamicTextReloadTexts();
			dwState := TLU.GetText(scReportMetaData.stReportTextList,scReportMetaData.stReportTxtId,ADR(stTempText),SIZEOF(stTempText)-SIZEOF(scReportMetaData.stAdditionalText));
			xFirstTryTextLoadLanguage := TRUE;
		END_IF; 
		(* Concat Additional Text to Repor*)
		IF scReportMetaData.stAdditionalText <> '' THEN
			stTempText := CONCAT(stTempText,CONCAT(' ',scReportMetaData.stAdditionalText));
		END_IF;		
	END_IF;
    (* Write Text to Output*)
    GetReportTextLanguage := stTempText;
END_METHOD

END_FUNCTION_BLOCK

// 30 Program Organization Units/OBJ/fcWordToHexString
FUNCTION fcWordToHexString : STRING[8]
VAR_INPUT
	wReportId		:	WORD;
END_VAR
VAR
	uiData		    :   UINT;
    uiDiv4          :   UINT;
    uiDiv3          :   UINT;
    uiDiv2          :   UINT;
    uiDiv1          :   UINT;
    uiPos4          :   UINT;                // 0-F
    uiPos3          :   UINT;                // 0-F
    uiPos2          :   UINT;                // 0-F
    uiPos1          :   UINT;                // 0-F    
    ayOfStr         :   ARRAY[0..15] OF STRING[1] := ['0','1','2','3','4','5','6','7','8','9','A','B','C','D','E','F'];
END_VAR

uiData := WORD_TO_UINT(wReportId);
IF uiData > 0 THEN
    uiPos4 :=                                                                  (uiData MOD (16));
    uiDiv4 :=                                  			        (uiData -(uiData MOD (16)))/(16);
    uiPos3 :=                                                                  (uiDiv4 MOD (16));
    uiDiv3 :=                                       		  (uiDiv4 - (uiDiv4  MOD (16)))/(16);
    uiPos2 :=                                                                  (uiDiv3 MOD (16));
    uiDiv2 :=                     						      (uiDiv3 - (uiDiv3  MOD (16)))/(16);        
    uiPos1 :=                                                                  (uiDiv2 MOD (16));

fcWordToHexString	 := CONCAT('16#',
                        CONCAT(ayOfStr[uiPos1],
                        CONCAT(ayOfStr[uiPos2],
                        CONCAT(ayOfStr[uiPos3],
                               ayOfStr[uiPos4]))));

ELSE
    fcWordToHexString := '16#0000';
END_IF;

END_FUNCTION

// 30 Program Organization Units/REPORTER/fbReportManager
FUNCTION_BLOCK FINAL fbReportManager IMPLEMENTS ITF_REPORTMANAGER
VAR_INPUT
	stErrorInitReportTextListIn 	:	POINTER TO stReportTextList;	
	stWarningInitReportTextListIn 	:	POINTER TO stReportTextList;	
	stInfoInitReportTextListIn 		:	POINTER TO stReportTextList;	
	scReportNr  					:	REFERENCE TO scReportNr;
END_VAR
VAR
	_stErrorReportTextListVis	    :	POINTER TO stReportTextList;	
	_stWarningReportTextListVis     :	POINTER TO stReportTextList;	
	_stInfoReportTextListVis 	    :	POINTER TO stReportTextList;	
	_stZusatzError					:	STRING(20);
	_stZusatzWarning				:	STRING(20);
	_stZusatzInfo					:	STRING(20);	
	xInitDone					    :	BOOL;	
    iAnzError                       :   INT;
    iAnzWarning                     :   INT;
    iAnzInfo                        :   INT;
END_VAR

PROPERTY proWarningText : STRING[100]
GET
VAR
	stReportTextList : stReportTextList;
	stIndex		 	 : STRING[3];
	stTempText		 : STRING[100];
END_VAR
IF _stWarningReportTextListVis <> 0 AND __ISVALIDREF(scReportNr) THEN 
	stIndex			 := TO_STRING(scReportNr.iWarning);
	TLU.GetText(_stWarningReportTextListVis^,stIndex,ADR(stTempText),SIZEOF(stTempText)-SIZEOF(_stZusatzWarning));
	proWarningText	 := Standard.CONCAT(stTempText,_stZusatzWarning);
ELSE
	proWarningText 	 := '';
END_IF;
END_GET
END_PROPERTY

METHOD metSyncReporter : BOOL
VAR_INPUT
	refFbReporter	:	REFERENCE TO fbReporter;
END_VAR
actInit();
IF __ISVALIDREF(refFbReporter) AND_THEN __ISVALIDREF(scReportNr) THEN
	(* Neuste Meldung Setzen *)
	IF refFbReporter.proNewReport THEN
        IF refFbReporter._enReportType = enReportType.Error THEN
            iAnzError                   := LIMIT(0,iAnzError + 1,32735);
        ELSIF refFbReporter._enReportType = enReportType.Warning THEN
            iAnzWarning                 := LIMIT(0,iAnzWarning + 1,32735);   
        ELSIF refFbReporter._enReportType = enReportType.Info THEN
            iAnzInfo                    := LIMIT(0,iAnzInfo + 1,32735);
        END_IF;  
        refFbReporter.proNewReport  := FALSE;  
    END_IF;   
    (* Aktive Meldung aktualisieren *)
    IF refFbReporter.proAktivReport THEN
        IF refFbReporter._enReportType = enReportType.Error THEN
            IF (scReportNr.iError = refFbReporter._iReportID OR scReportNr.iError = 0) OR scReportNr.usiErrorPrio = 0 OR (scReportNr.usiErrorPrio >= refFbReporter.proPrio AND refFbReporter.proPrio > 0) THEN
                    scReportNr.iError           := refFbReporter._iReportID;
                    scReportNr.usiErrorPrio     := refFbReporter.usiPrio; 
                    _stErrorReportTextListVis   := refFbReporter._stReportTextList;
					_stZusatzError				:= refFbReporter.proOptionalText;
					refFbReporter.proNewReport  := FALSE;   
             END_IF;
        ELSIF refFbReporter._enReportType = enReportType.Warning THEN
            IF (scReportNr.iWarning = refFbReporter._iReportID OR scReportNr.iWarning = 0) OR scReportNr.usiWarnungPrio = 0 OR  (scReportNr.usiWarnungPrio >= refFbReporter.proPrio AND refFbReporter.proPrio > 0) THEN
                scReportNr.iWarning         := refFbReporter._iReportID;
                scReportNr.usiWarnungPrio   := refFbReporter.usiPrio;
                _stWarningReportTextListVis := refFbReporter._stReportTextList;
				_stZusatzWarning				:= refFbReporter.proOptionalText;
                refFbReporter.proNewReport  := FALSE;   
            END_IF;
        ELSIF refFbReporter._enReportType = enReportType.Info THEN
            IF (scReportNr.iInfo = refFbReporter._iReportID OR scReportNr.iInfo = 0) OR scReportNr.usiInfoPrio = 0 OR (scReportNr.usiInfoPrio >= refFbReporter.proPrio AND refFbReporter.proPrio > 0) THEN
                scReportNr.iInfo            := refFbReporter._iReportID;
                scReportNr.usiInfoPrio      := refFbReporter.usiPrio;
                _stInfoReportTextListVis    := refFbReporter._stReportTextList;
				_stZusatzInfo				:= refFbReporter.proOptionalText;
                refFbReporter.proNewReport  := FALSE;	        		
            END_IF;
        END_IF;
    END_IF;
	(* Inaktive Meldung rücksetzten *)
	IF NOT refFbReporter.proAktivReport THEN
		IF refFbReporter._enReportType = enReportType.Error AND_THEN scReportNr.iError = refFbReporter._iReportID THEN
			scReportNr.iError           := 0;
            scReportNr.usiErrorPrio     := 0;
			_stErrorReportTextListVis   := stErrorInitReportTextListIn;
		ELSIF refFbReporter._enReportType = enReportType.Warning AND_THEN scReportNr.iWarning = refFbReporter._iReportID THEN
			scReportNr.iWarning         := 0;
            scReportNr.usiWarnungPrio   := 0;
			_stWarningReportTextListVis := stWarningInitReportTextListIn;
		ELSIF refFbReporter._enReportType = enReportType.Info AND_THEN scReportNr.iInfo = refFbReporter._iReportID THEN
			scReportNr.iInfo            := 0;
            scReportNr.usiInfoPrio      := 0;
			_stInfoReportTextListVis    := stInfoInitReportTextListIn;		
		END_IF;	
	END_IF;	
	(* Counter Done *)
	IF refFbReporter.proDoneReport THEN
		IF refFbReporter._enReportType = enReportType.Error THEN
            iAnzError                       := LIMIT(0,iAnzError - 1,32735);
		ELSIF refFbReporter._enReportType = enReportType.Warning THEN
            iAnzWarning                     := LIMIT(0,iAnzWarning - 1,32735);
		ELSIF refFbReporter._enReportType = enReportType.Info THEN
            iAnzInfo                        :=LIMIT(0,iAnzInfo - 1,32735);
		END_IF;	
        refFbReporter.proDoneReport     := FALSE;
	END_IF;				
END_IF
END_METHOD

PROPERTY proInfoText : STRING[100]
GET
VAR
	stReportTextList : stReportTextList;
	stIndex		 	 : STRING[3];
	stTempText		 : STRING[100];
END_VAR
IF _stInfoReportTextListVis <> 0 AND __ISVALIDREF(scReportNr) THEN 
	stIndex			:= TO_STRING(scReportNr.iInfo);
	TLU.GetText(_stInfoReportTextListVis^,stIndex,ADR(stTempText),SIZEOF(stTempText)-SIZEOF(_stZusatzInfo));
	proInfoText	 := Standard.CONCAT(stTempText,_stZusatzInfo);
ELSE
	proInfoText := '';
END_IF;
END_GET
END_PROPERTY

PROPERTY proErrorText : STRING[100]
GET
VAR
	stIndex		 	 : STRING[3];
	stTempText		 : STRING[100];
END_VAR
IF _stErrorReportTextListVis <> 0 AND __ISVALIDREF(scReportNr) THEN 
	stIndex			:= TO_STRING(scReportNr.iError);
	TLU.GetText(_stErrorReportTextListVis^,stIndex,ADR(stTempText),SIZEOF(stTempText)-SIZEOF(_stZusatzError));
	proErrorText	 := Standard.CONCAT(stTempText,_stZusatzError);
ELSE
	proErrorText := '';
END_IF;
END_GET
END_PROPERTY

PROPERTY proGetErrorNr : INT
GET
IF __ISVALIDREF(scReportNr) THEN
    proGetErrorNr := scReportNr.iError;
ELSE
    proGetErrorNr := 0;
END_IF;
END_GET
END_PROPERTY

ACTION actInit:
IF NOT xInitDone AND_THEN stErrorInitReportTextListIn <> 0
				 AND_THEN stWarningInitReportTextListIn <> 0
				 AND_THEN stInfoInitReportTextListIn <> 0 THEN 
	_stErrorReportTextListVis 	:= stErrorInitReportTextListIn;
	_stWarningReportTextListVis	:= stWarningInitReportTextListIn;
	_stInfoReportTextListVis	:= stInfoInitReportTextListIn;
	xInitDone := TRUE;
END_IF;
END_ACTION

PROPERTY proGetWarningNr : INT
GET
IF __ISVALIDREF(scReportNr) THEN
    proGetWarningNr := scReportNr.iWarning;
ELSE
    proGetWarningNr := 0;
END_IF;
END_GET
END_PROPERTY

PROPERTY proGetInfoNr : INT
GET
IF __ISVALIDREF(scReportNr) THEN
    proGetInfoNr := scReportNr.iInfo;
ELSE
    proGetInfoNr := 0;
END_IF;
END_GET
END_PROPERTY

PROPERTY proAnzError : INT
GET
proAnzError := iAnzError;
END_GET
END_PROPERTY

PROPERTY proAnzWarning : INT
GET
proAnzWarning := iAnzWarning;
END_GET
END_PROPERTY

PROPERTY proAnzInfo : INT
GET
proAnzInfo:= iAnzInfo;
END_GET
END_PROPERTY

PROPERTY proTotalReports : INT
GET
proTotalReports := iAnzInfo + iAnzWarning + iAnzError;
END_GET
END_PROPERTY

END_FUNCTION_BLOCK

// 40 Visualizations/REPORT_ID
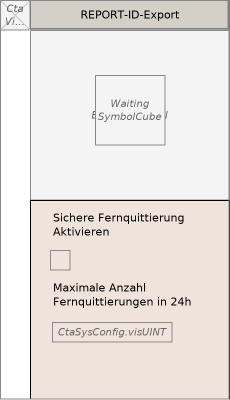
VISUALIZATION REPORT_ID  // 230x400
VAR_IN_OUT
    iPos    :INT;	
    fbReportVisuIn        :   fbReportVisu; 
END_VAR
    Rectangle (30,0 200x200)
    Rectangle (0,0 230x30)
    Button (30,0 200x30), "REPORT-ID-Export", pressed state: GVL_Report.fbDataHandler.proExport
        tap GVL_Report.fbDataHandler.proExportIdStart
    BrowserControl (30,30 200x170)
        p3734058945: 'History/IDDownload.htm'
        p2179181546: GVL_Report.fbDataHandler.xExportDone
    Image (0,0 30x30), image: CtaVisSymbols.ImagePool.arrow-right_solo_black
        OnMouseClick: execute { iPos := 0; }
    Rectangle (30,200 200x199)
    Label (50,280 168x30), "Maximale Anzahl Fernquittierungen in 24h"
    Frame (52,322 120x20)
        shows CtaSysConfig.visUINT(visfbUINTIn := fbReportVisuIn.scPara.fbuiMaxFernQuitt)
    Frame (50,250 20x20)
        shows CtaSysConfig.visBOOL(visfbBOOLIn := fbReportVisuIn.scPara.fbxEnSafetyFernQuitt)
    Label (50,210 168x30), "Sichere Fernquittierung Aktivieren"
    WaitingSymbolCube (95,75 70x70), invisible if: NOT GVL_Report.fbDataHandler.proExport
END_VISUALIZATION

// 40 Visualizations/TABLE/VIS_REPORT_TABLE
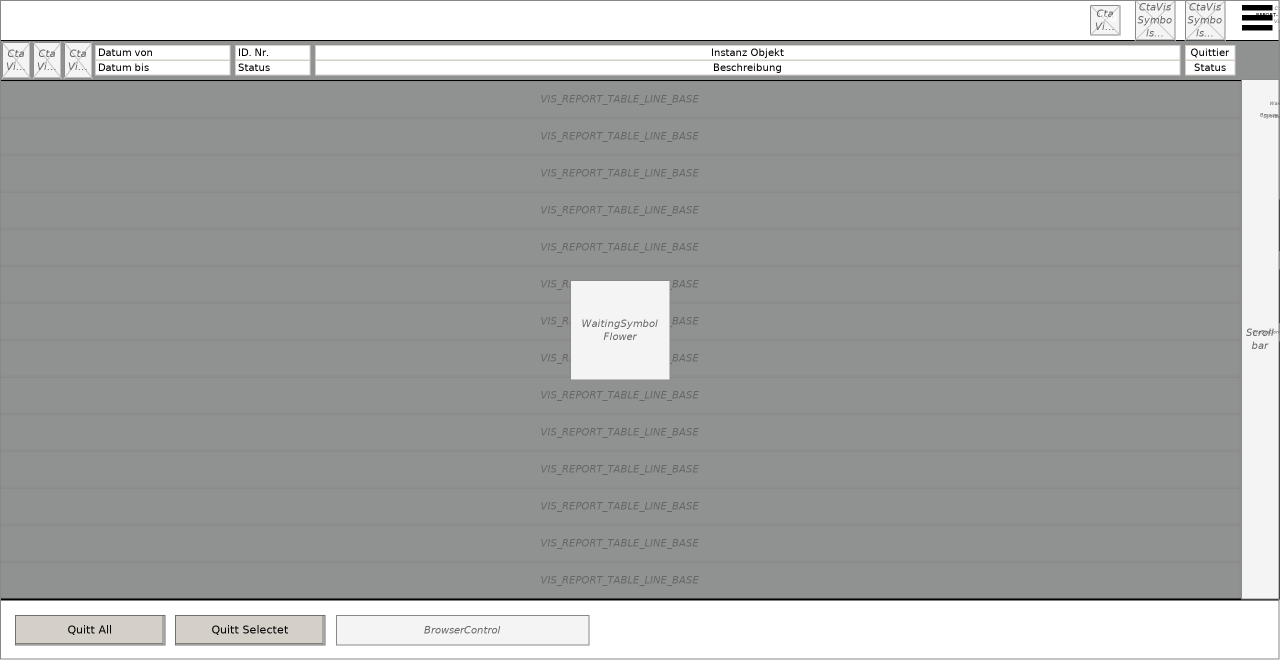
VISUALIZATION VIS_REPORT_TABLE  // 1280x660
    Frame (0,0 1280x660)
        shows VIS_REPORT_TABLE_BASE(fbReportVisuIn := GVL_Report.fbReportVisu)
END_VISUALIZATION

// 40 Visualizations/PUSHLINE/VIS_REPORT_PUSH_LINE
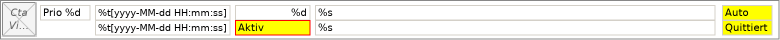
VISUALIZATION VIS_REPORT_PUSH_LINE  // 780x40
    Frame (0,0 780x40), invisible if: GVL_Report.fbReportObjectFactory.proGetAktiveReport = 0
        shows VIS_REPORT_PUSH_LINE_QUERRY()
END_VISUALIZATION

// 40 Visualizations/PUSHLINE/VIS_REPORT_PUSH_LINE_BASE
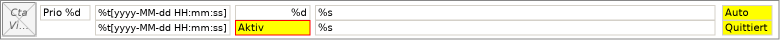
VISUALIZATION VIS_REPORT_PUSH_LINE_BASE  // 780x40
VAR_INPUT
    ITF_REPORTOBJECT_VIS : ITF_REPORTOBJECT;	
END_VAR
    Textfield (235,5 75x15), "%d", text variable: ITF_REPORTOBJECT_VIS.proReportId
    Image (2,2 34x34), invisible if: ITF_REPORTOBJECT_VIS.proReportType <> enReportType.Error, image: CtaVisSymbols.ImagePool.CtaError
    Textfield (95,5 135x15), "%t[yyyy-MM-dd HH:mm:ss]", text variable: ITF_REPORTOBJECT_VIS.proDtFrom, invisible if: ITF_REPORTOBJECT_VIS.proDtFrom = TO_DT(0)
    Textfield (315,5 400x15), "%s", text variable: ITF_REPORTOBJECT_VIS.proGetReporterText
    Textfield (315,20 400x15), "%s", text variable: ITF_REPORTOBJECT_VIS.proGetReportText
    Textfield (95,20 135x15), "%t[yyyy-MM-dd HH:mm:ss]", text variable: ITF_REPORTOBJECT_VIS.proDtTo, invisible if: ITF_REPORTOBJECT_VIS.proDtTo = TO_DT(0)
    Textfield (40,5 50x15), "Prio %d", text variable: ITF_REPORTOBJECT_VIS.proPrio
    Textfield (235,20 75x15), "Aktiv", colour toggle: ITF_REPORTOBJECT_VIS.proReportIn, invisible if: NOT ITF_REPORTOBJECT_VIS.proStateActive
    Textfield (722,20 50x15), "Quittiert", colour toggle: ITF_REPORTOBJECT_VIS.proIsQuitt AND NOT ITF_REPORTOBJECT_VIS.proStateActive, invisible if: NOT ITF_REPORTOBJECT_VIS.proIsQuitt
    Image (2,2 34x34), invisible if: ITF_REPORTOBJECT_VIS.proReportType <> enReportType.Info, image: CtaVisSymbols.ImagePool.CtaInfo
    Image (2,2 34x34), invisible if: ITF_REPORTOBJECT_VIS.proReportType <> enReportType.Warning, image: CtaVisSymbols.ImagePool.CtaWarning
    Textfield (722,5 50x15), "Auto", colour toggle: ITF_REPORTOBJECT_VIS.proIsQuitt AND NOT ITF_REPORTOBJECT_VIS.proStateActive, invisible if: ITF_REPORTOBJECT_VIS.proReportAcknowledgType <> enReportacknowledgeType.Auto OR NOT ITF_REPORTOBJECT_VIS.proIsQuitt
END_VISUALIZATION

// 40 Visualizations/PUSHLINE/VIS_REPORT_PUSH_LINE_QUERRY
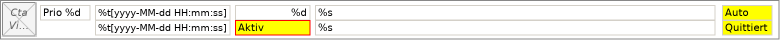
VISUALIZATION VIS_REPORT_PUSH_LINE_QUERRY  // 780x40
    Frame (0,0 780x40)
        shows VIS_REPORT_PUSH_LINE_BASE(ITF_REPORTOBJECT_VIS := GVL_Report.fbReportObjectFactory.proGetAktiveReport)
END_VISUALIZATION

// 40 Visualizations/REPORTMANAGER/VIS_REPORTMANAGER
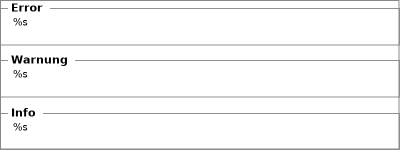
VISUALIZATION VIS_REPORTMANAGER  // 400x150
VAR_INPUT
    ITF_REPORTMANAGER : ITF_REPORTMANAGER;	  
END_VAR
    Frame (0,0 400x150), invisible if: ITF_REPORTMANAGER = 0
        shows VIS_REPORTMANAGER_BASE(ITF_REPORTMANAGER := ITF_REPORTMANAGER)
END_VISUALIZATION

// 40 Visualizations/TABLE LINE/VIS_REPORT_TABLE_LINE_BASE
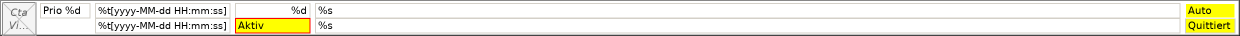
VISUALIZATION VIS_REPORT_TABLE_LINE_BASE  // 1240x36
VAR_INPUT
    ITF_REPORTOBJECT_VIS : ITF_REPORTOBJECT;	
END_VAR
    RoundedRectangle (0,0 1240x36)
    Textfield (235,3 75x15), "%d", text variable: ITF_REPORTOBJECT_VIS.proReportId
    Textfield (95,18 135x15)
    Textfield (95,3 135x15)
    Image (2,2 34x34), invisible if: ITF_REPORTOBJECT_VIS.proReportType <> enReportType.Error, image: CtaVisSymbols.ImagePool.CtaError
    Textfield (95,3 135x15), "%t[yyyy-MM-dd HH:mm:ss]", text variable: ITF_REPORTOBJECT_VIS.proDtFrom, invisible if: ITF_REPORTOBJECT_VIS.proDtFrom = TO_DT(0)
    Textfield (315,3 865x15), "%s", text variable: ITF_REPORTOBJECT_VIS.proGetReporterText
    Textfield (315,18 865x15), "%s", text variable: ITF_REPORTOBJECT_VIS.proGetReportText
    Textfield (95,18 135x15), "%t[yyyy-MM-dd HH:mm:ss]", text variable: ITF_REPORTOBJECT_VIS.proDtTo, invisible if: ITF_REPORTOBJECT_VIS.proDtTo = TO_DT(0)
    Textfield (40,3 50x15), "Prio %d", text variable: ITF_REPORTOBJECT_VIS.proPrio
    Textfield (235,18 75x15), "Aktiv", colour toggle: ITF_REPORTOBJECT_VIS.proReportIn, invisible if: NOT ITF_REPORTOBJECT_VIS.proStateActive
    Textfield (1185,18 50x15), "Quittiert", colour toggle: ITF_REPORTOBJECT_VIS.proIsQuitt AND NOT ITF_REPORTOBJECT_VIS.proStateActive, invisible if: NOT ITF_REPORTOBJECT_VIS.proIsQuitt
    Image (2,2 34x34), invisible if: ITF_REPORTOBJECT_VIS.proReportType <> enReportType.Info, image: CtaVisSymbols.ImagePool.CtaInfo
    Image (2,2 34x34), invisible if: ITF_REPORTOBJECT_VIS.proReportType <> enReportType.Warning, image: CtaVisSymbols.ImagePool.CtaWarning
    Textfield (1185,3 50x15), "Auto", colour toggle: ITF_REPORTOBJECT_VIS.proIsQuitt AND NOT ITF_REPORTOBJECT_VIS.proStateActive, invisible if: ITF_REPORTOBJECT_VIS.proReportAcknowledgType <> enReportacknowledgeType.Auto OR NOT ITF_REPORTOBJECT_VIS.proIsQuitt
    RoundedRectangle (0,0 1240x36), colour toggle: ITF_REPORTOBJECT_VIS.proIsSelected
        OnMouseClick: execute { ITF_REPORTOBJECT_VIS.proIsSelected := NOT ITF_REPORTOBJECT_VIS.proIsSelected; }
END_VISUALIZATION

// 40 Visualizations/REPORTMANAGER/VIS_REPORTMANAGER_BASE
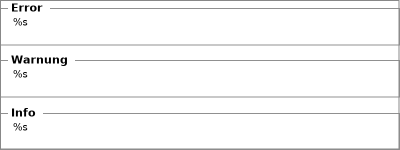
VISUALIZATION VIS_REPORTMANAGER_BASE  // 400x150
VAR_INPUT
    ITF_REPORTMANAGER : ITF_REPORTMANAGER;	  
END_VAR
    GroupBox (0,52 400x45), "Warnung"
        Textfield (10,15 380x30), "%s", text variable: ITF_REPORTMANAGER.proWarningText, text list: ''
    GroupBox (0,105 400x45), "Info"
        Textfield (10,15 380x30), "%s", text variable: ITF_REPORTMANAGER.proInfoText, text list: ''
    GroupBox (0,0 400x45), "Error"
        Textfield (10,15 380x30), "%s", text variable: ITF_REPORTMANAGER.proErrorText, text list: ''
END_VISUALIZATION

// 40 Visualizations/TABLE/VIS_REPORT_TABLE_BASE
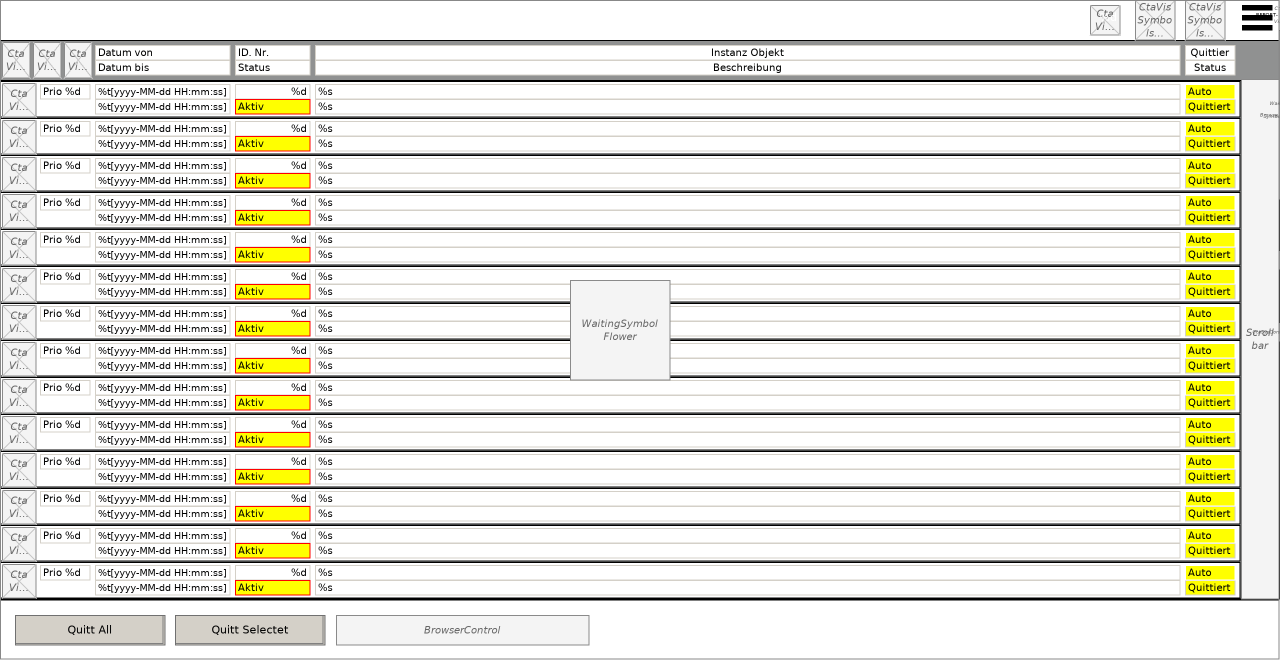
VISUALIZATION VIS_REPORT_TABLE_BASE  // 1280x660
VAR_IN_OUT
    fbReportVisuIn        :   fbReportVisu;     
END_VAR
VAR
    iPos            :   INT;
    xRefresh        :   BOOL;
END_VAR
    Rectangle (0,40 1279x560)
    Rectangle (0,80 1280x519)
    Frame (0,414 1240x36), invisible if: NOT fbReportVisuIn.metGetShowReport(9,CurrentClientId), input disabled if: fbReportVisuIn.ayenVisuTableType[CurrentClientId] = enTableType.HISTORY_REPORTS
        shows VIS_REPORT_TABLE_LINE(ITF_REPORTOBJECT_VIS := fbReportVisuIn.metGetReport(9,CurrentClientId))
    Frame (0,377 1240x36), invisible if: NOT fbReportVisuIn.metGetShowReport(8,CurrentClientId), input disabled if: fbReportVisuIn.ayenVisuTableType[CurrentClientId] = enTableType.HISTORY_REPORTS
        shows VIS_REPORT_TABLE_LINE(ITF_REPORTOBJECT_VIS := fbReportVisuIn.metGetReport(8,CurrentClientId))
    Frame (0,340 1240x36), invisible if: NOT fbReportVisuIn.metGetShowReport(7,CurrentClientId), input disabled if: fbReportVisuIn.ayenVisuTableType[CurrentClientId] = enTableType.HISTORY_REPORTS
        shows VIS_REPORT_TABLE_LINE(ITF_REPORTOBJECT_VIS := fbReportVisuIn.metGetReport(7,CurrentClientId))
    Frame (0,303 1240x36), invisible if: NOT fbReportVisuIn.metGetShowReport(6,CurrentClientId), input disabled if: fbReportVisuIn.ayenVisuTableType[CurrentClientId] = enTableType.HISTORY_REPORTS
        shows VIS_REPORT_TABLE_LINE(ITF_REPORTOBJECT_VIS := fbReportVisuIn.metGetReport(6,CurrentClientId))
    Frame (0,266 1240x36), invisible if: NOT fbReportVisuIn.metGetShowReport(5,CurrentClientId), input disabled if: fbReportVisuIn.ayenVisuTableType[CurrentClientId] = enTableType.HISTORY_REPORTS
        shows VIS_REPORT_TABLE_LINE(ITF_REPORTOBJECT_VIS := fbReportVisuIn.metGetReport(5,CurrentClientId))
    Frame (0,229 1240x36), invisible if: NOT fbReportVisuIn.metGetShowReport(4,CurrentClientId), input disabled if: fbReportVisuIn.ayenVisuTableType[CurrentClientId] = enTableType.HISTORY_REPORTS
        shows VIS_REPORT_TABLE_LINE(ITF_REPORTOBJECT_VIS := fbReportVisuIn.metGetReport(4,CurrentClientId))
    Frame (0,192 1240x36), invisible if: NOT fbReportVisuIn.metGetShowReport(3,CurrentClientId), input disabled if: fbReportVisuIn.ayenVisuTableType[CurrentClientId] = enTableType.HISTORY_REPORTS
        shows VIS_REPORT_TABLE_LINE(ITF_REPORTOBJECT_VIS := fbReportVisuIn.metGetReport(3,CurrentClientId))
    Frame (0,155 1240x36), invisible if: NOT fbReportVisuIn.metGetShowReport(2,CurrentClientId), input disabled if: fbReportVisuIn.ayenVisuTableType[CurrentClientId] = enTableType.HISTORY_REPORTS
        shows VIS_REPORT_TABLE_LINE(ITF_REPORTOBJECT_VIS := fbReportVisuIn.metGetReport(2,CurrentClientId))
    Frame (0,118 1240x36), invisible if: NOT fbReportVisuIn.metGetShowReport(1,CurrentClientId), input disabled if: fbReportVisuIn.ayenVisuTableType[CurrentClientId] = enTableType.HISTORY_REPORTS
        shows VIS_REPORT_TABLE_LINE(ITF_REPORTOBJECT_VIS := fbReportVisuIn.metGetReport(1,CurrentClientId))
    Frame (0,81 1240x36), invisible if: NOT fbReportVisuIn.metGetShowReport(0,CurrentClientId), input disabled if: fbReportVisuIn.ayenVisuTableType[CurrentClientId] = enTableType.HISTORY_REPORTS
        shows VIS_REPORT_TABLE_LINE(ITF_REPORTOBJECT_VIS := fbReportVisuIn.metGetReport(0,CurrentClientId))
    Group (1242,5 35x25)
        OnMouseClick: execute { iPos := -230; }
        RoundedRectangle (0,0 30x5)
        RoundedRectangle (0,10 30x5)
        RoundedRectangle (0,20 30x5)
    Textfield (95,45 135x15), "Datum von"
    Textfield (95,60 135x15), "Datum bis"
    Textfield (235,45 75x15), "ID. Nr."
    Textfield (235,60 75x15), "Status"
    Textfield (315,45 865x15), "Instanz Objekt"
    Textfield (315,60 865x15), "Beschreibung"
    Textfield (1185,45 50x15), "Quittier"
    Textfield (1185,60 50x15), "Status"
    Group (15,615 310x30)
        Button (0,0 150x30), "Quitt All"
            OnMouseClick: execute { GVL_Report.fbReportObjectFactory.metQuittAllReports(); }
        Button (160,0 150x30), "Quitt Selectet", invisible if: fbReportVisuIn.ayenVisuTableType[CurrentClientId] = enTableType.HISTORY_REPORTS
            OnMouseClick: execute { GVL_Report.fbReportObjectFactory.metQuittSelectedReports(); }
    Group (63,41 30x38)
        OnMouseClick: execute { fbReportVisuIn.FilterInfo(NOT fbReportVisuIn.ayFilterInfo[CurrentClientId],CurrentClientID); }
        Image (1,1 28x36), invisible if: fbReportVisuIn.ayenVisuTableType[CurrentClientId] = enTableType.HISTORY_REPORTS, image: CtaVisSymbols.ImagePool.CtaInfo
        Rectangle (0,0 30x38), colour toggle: fbReportVisuIn.ayFilterInfo[CurrentClientId], invisible if: fbReportVisuIn.ayenVisuTableType[CurrentClientId] = enTableType.HISTORY_REPORTS
            OnMouseClick: execute { fbReportVisuIn.FilterInfo(NOT fbReportVisuIn.ayFilterInfo[CurrentClientId],CurrentClientID); }
    Group (32,41 30x38)
        OnMouseClick: execute { fbReportVisuIn.FilterWarning(NOT fbReportVisuIn.ayFilterWarning[CurrentClientId],CurrentClientID); }
        Image (1,1 28x36), invisible if: fbReportVisuIn.ayenVisuTableType[CurrentClientId] = enTableType.HISTORY_REPORTS, image: CtaVisSymbols.ImagePool.CtaWarning
            OnMouseClick: execute { fbReportVisuIn.FilterWarning(NOT fbReportVisuIn.ayFilterWarning[CurrentClientId],CurrentClientID); }
        Rectangle (0,0 30x38), colour toggle: fbReportVisuIn.ayFilterWarning[CurrentClientId], invisible if: fbReportVisuIn.ayenVisuTableType[CurrentClientId] = enTableType.HISTORY_REPORTS
            OnMouseClick: execute { fbReportVisuIn.FilterWarning(NOT fbReportVisuIn.ayFilterWarning[CurrentClientId],CurrentClientID); }
    Group (1,41 30x38)
        OnMouseClick: execute { fbReportVisuIn.FilterError(NOT fbReportVisuIn.ayFilterError[CurrentClientId],CurrentClientID); }
        Image (1,1 28x36), colour toggle: fbReportVisuIn.ayFilterError[CurrentClientId], invisible if: fbReportVisuIn.ayenVisuTableType[CurrentClientId] = enTableType.HISTORY_REPORTS, image: CtaVisSymbols.ImagePool.CtaError
            OnMouseClick: execute { fbReportVisuIn.FilterError(NOT fbReportVisuIn.ayFilterError[CurrentClientId],CurrentClientID); }
        Rectangle (0,0 30x38), colour toggle: fbReportVisuIn.ayFilterError[CurrentClientId], invisible if: fbReportVisuIn.ayenVisuTableType[CurrentClientId] = enTableType.HISTORY_REPORTS
            OnMouseClick: execute { fbReportVisuIn.FilterError(NOT fbReportVisuIn.ayFilterError[CurrentClientId],CurrentClientID); }
    Group (1085,0 40x40)
        Image (5,5 30x30), image: CtaVisSymbols.ImagePool.message
            OnMouseClick: execute { fbReportVisuIn.ayenVisuTableType[CurrentClientId] := enTableType.PENDING_REPORTS; fbReportVisuIn.ayOffset[CurrentClientId]		  := 0; }
        Rectangle (0,0 40x40), colour toggle: fbReportVisuIn.ayenVisuTableType[CurrentClientId] = enTableType.PENDING_REPORTS
            OnMouseClick: execute { fbReportVisuIn.ayenVisuTableType[CurrentClientId] := enTableType.PENDING_REPORTS; fbReportVisuIn.ayOffset[CurrentClientId] := 0; }
        Textfield (5,10 30x15), "%d", text variable: fbReportVisuIn.proAnzReportsInTable, invisible if: fbReportVisuIn.proAnzReportsInTable = 0
            OnMouseClick: execute { fbReportVisuIn.ayenVisuTableType[CurrentClientId] := enTableType.PENDING_REPORTS; fbReportVisuIn.ayOffset[CurrentClientId] := 0; }
    Scrollbar (1241,79 38x520), input disabled if: fbReportVisuIn.ayWaitToReload[CurrentClientId] > 0 AND fbReportVisuIn.ayWaitToReload[CurrentClientId] < 3
        p2245068023: fbReportVisuIn.MaxOffset(CurrentClientId)
        p1057716461: fbReportVisuIn.ayOffset[CurrentClientId]
    Group (1135,0 40x40)
        Image (0,0 40x40), image: CtaVisSymbols.ImagePool.database_black
            OnMouseClick: execute { fbReportVisuIn.ayenVisuTableType[CurrentClientId] := enTableType.HISTORY_REPORTS; fbReportVisuIn.ayOffset[CurrentClientId] := 0; }
        Rectangle (0,0 40x40), colour toggle: fbReportVisuIn.ayenVisuTableType[CurrentClientId] = enTableType.HISTORY_REPORTS
            OnMouseClick: execute { fbReportVisuIn.ayenVisuTableType[CurrentClientId] := enTableType.HISTORY_REPORTS; fbReportVisuIn.ayOffset[CurrentClientId] := 0; }
    Group (1185,0 40x40), invisible if: fbReportVisuIn.ayenVisuTableType[CurrentClientId] = enTableType.PENDING_REPORTS
        OnMouseClick:  Dialog=VIS_REPORT_DELETE, OpenModal=True, OpenCentered=True
        Image (0,0 40x40), invisible if: fbReportVisuIn.ayenVisuTableType[CurrentClientId] = enTableType.PENDING_REPORTS, image: CtaVisSymbols.ImagePool.delete_solo_black
        Rectangle (0,0 40x40), invisible if: fbReportVisuIn.ayenVisuTableType[CurrentClientId] = enTableType.PENDING_REPORTS
    BrowserControl (336,615 253x30), invisible if: fbReportVisuIn.ayenVisuTableType[CurrentClientId] = enTableType.PENDING_REPORTS
        p3734058945: 'History/HistoryDownload.htm'
        p2179181546: fbReportVisuIn.ayenVisuTableType[CurrentClientId] = enTableType.HISTORY_REPORTS
    Frame (0,451 1240x36), invisible if: NOT fbReportVisuIn.metGetShowReport(10,CurrentClientId), input disabled if: fbReportVisuIn.ayenVisuTableType[CurrentClientId] = enTableType.HISTORY_REPORTS
        shows VIS_REPORT_TABLE_LINE(ITF_REPORTOBJECT_VIS := fbReportVisuIn.metGetReport(10,CurrentClientId))
    Frame (0,488 1240x36), invisible if: NOT fbReportVisuIn.metGetShowReport(11,CurrentClientId), input disabled if: fbReportVisuIn.ayenVisuTableType[CurrentClientId] = enTableType.HISTORY_REPORTS
        shows VIS_REPORT_TABLE_LINE(ITF_REPORTOBJECT_VIS := fbReportVisuIn.metGetReport(11,CurrentClientId))
    Frame (0,525 1240x36), invisible if: NOT fbReportVisuIn.metGetShowReport(12,CurrentClientId), input disabled if: fbReportVisuIn.ayenVisuTableType[CurrentClientId] = enTableType.HISTORY_REPORTS
        shows VIS_REPORT_TABLE_LINE(ITF_REPORTOBJECT_VIS := fbReportVisuIn.metGetReport(12,CurrentClientId))
    Frame (0,562 1240x36), invisible if: NOT fbReportVisuIn.metGetShowReport(13,CurrentClientId), input disabled if: fbReportVisuIn.ayenVisuTableType[CurrentClientId] = enTableType.HISTORY_REPORTS
        shows VIS_REPORT_TABLE_LINE(ITF_REPORTOBJECT_VIS := fbReportVisuIn.metGetReport(13,CurrentClientId))
    Frame (1279,0 0x400), invisible if: iPos = 0
        shows REPORT_ID(iPos := iPos, fbReportVisuIn := fbReportVisuIn)
        p3560616238: iPos
        p874137650: iPos * -1
    WaitingSymbolFlower (570,280 100x100), invisible if: fbReportVisuIn.ayWaitToReload[CurrentClientId] = 0 OR fbReportVisuIn.ayWaitToReload[CurrentClientId] = 3
END_VISUALIZATION

// 40 Visualizations/TABLE LINE/VIS_REPORT_TABLE_LINE_QUERRY
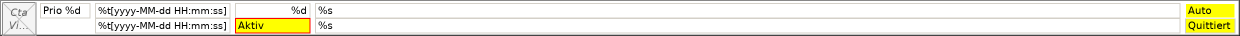
VISUALIZATION VIS_REPORT_TABLE_LINE_QUERRY  // 1240x36
VAR_INPUT
    ITF_REPORTOBJECT_VIS : ITF_REPORTOBJECT;	
END_VAR
    Frame (0,0 1240x36), invisible if: NOT __QUERYINTERFACE(ITF_REPORTOBJECT_VIS,ITF_REPORTOBJECT_VIS)
        shows VIS_REPORT_TABLE_LINE_BASE(ITF_REPORTOBJECT_VIS := ITF_REPORTOBJECT_VIS)
END_VISUALIZATION

// 40 Visualizations/TABLE LINE/VIS_REPORT_TABLE_LINE
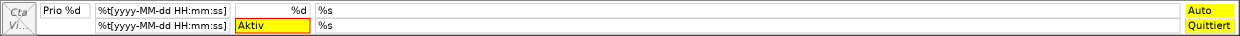
VISUALIZATION VIS_REPORT_TABLE_LINE  // 1240x36
VAR_INPUT
    ITF_REPORTOBJECT_VIS : ITF_REPORTOBJECT;	
END_VAR
    Frame (0,0 1240x36), invisible if: NOT __QUERYINTERFACE(ITF_REPORTOBJECT_VIS,ITF_REPORTOBJECT_VIS)
        shows VIS_REPORT_TABLE_LINE_QUERRY(ITF_REPORTOBJECT_VIS := ITF_REPORTOBJECT_VIS)
END_VISUALIZATION

// 40 Visualizations/HAND/VIS_REPORT_HAND
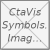
VISUALIZATION VIS_REPORT_HAND  // 50x50
    Image (0,0 50x50), invisible if: GVL_Report.diCountHand = 0, image: CtaVisSymbols.ImagePool.front_hand_Yellow
END_VISUALIZATION

// 40 Visualizations/TABLE/DELETE/VIS_REPORT_DELETE
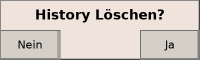
VISUALIZATION VIS_REPORT_DELETE  // 200x60
    Rectangle (0,0 200x60)
    Button (140,30 60x30), "Ja"
        OnMouseClick: execute { GVL_Report.fbDataHandler.metDeleteHistory(); }
        OnMouseClick:  Dialog=VIS_REPORT_DELETE, Result=Yes, NumpadKeypadSet=True
    Button (0,30 60x30), "Nein"
        OnMouseClick:  Dialog=VIS_REPORT_DELETE, Result=No, NumpadKeypadSet=True
    Label (0,0 200x30), "History Löschen?"
END_VISUALIZATION

// 40 Visualizations/ANZAHL REPORTS/Modul/VIS_ANZ_REPORTS_MODUL
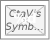
VISUALIZATION VIS_ANZ_REPORTS_MODUL  // 50x40
VAR_IN_OUT
	ITF_REPORTMANAGER_IN	:	ITF_REPORTMANAGER;
END_VAR
    Frame (0,0 50x40), invisible if: NOT(__QUERYINTERFACE(ITF_REPORTMANAGER_IN,ITF_REPORTMANAGER_IN))
        shows VIS_ANZ_REPORTS_MODUL_QUERRY(ITF_REPORTMANAGER_IN := ITF_REPORTMANAGER_IN)
END_VISUALIZATION

// 40 Visualizations/ANZAHL REPORTS/VIS_ANZ_REPORTS_OVERALL
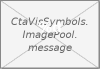
VISUALIZATION VIS_ANZ_REPORTS_OVERALL  // 100x69
    Image (0,0 100x69), image: CtaVisSymbols.ImagePool.message
    Textfield (35,20 30x15), "%d", text variable: GVL_Report.fbSort.proAnzAktiveReports, invisible if: GVL_Report.fbSort.proAnzAktiveReports = 0
END_VISUALIZATION

// 40 Visualizations/ANZAHL REPORTS/Modul/VIS_ANZ_REPORTS_MODUL_BASE
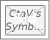
VISUALIZATION VIS_ANZ_REPORTS_MODUL_BASE  // 50x40
VAR_IN_OUT
	ITF_REPORTMANAGER_IN	:	ITF_REPORTMANAGER;
END_VAR
    Image (5,5 40x30), image: CtaVisSymbols.ImagePool.message
    Textfield (10,11 30x15), "%d", text variable: ITF_REPORTMANAGER_IN.proTotalReports, invisible if: ITF_REPORTMANAGER_IN.proTotalReports = 0
END_VISUALIZATION

// 40 Visualizations/ANZAHL REPORTS/Modul/VIS_ANZ_REPORTS_MODUL_QUERRY
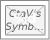
VISUALIZATION VIS_ANZ_REPORTS_MODUL_QUERRY  // 50x40
VAR_IN_OUT
	ITF_REPORTMANAGER_IN	:	ITF_REPORTMANAGER;
END_VAR
    Frame (0,0 50x40)
        shows VIS_ANZ_REPORTS_MODUL_BASE(ITF_REPORTMANAGER_IN := ITF_REPORTMANAGER_IN)
END_VISUALIZATION

(* text list txtLibAp99_1Error (id | default | de | en | fr | it)
  99 | Maximale Anzahl Fernquittierungen erreicht | Maximale Anzahl Fernquittierungen erreicht | Maximum number of remote acknowledgements reached | Nombre maximal d'acquittements à distance atteint | Raggiunto il numero massimo di conferme remote
   |  |  |  |  |  *)

(* text list txtLibAp99_2enTypeOfAck (id | default | de | en | fr | it)
  0 | Automatisch | Automatisch |  |  | 
  1 | Quittierpflicht | Quittierpflicht |  |  | 
  2 | Wiederholend bis N | Wiederholend bis N |  |  | 
   |  |  |  |  |  *)

(* text list txtLibAp99_2Warnung (id | default | de | en | fr | it)
  99 | Fernquittierung Erfolgt. Anzahl noch Mögliche Fernquittierungen: | Fernquittierung Erfolgt. Anzahl noch Mögliche Fernquittierungen: | Remote acknowledgement Done. Number of remote acknowledgements still possible: | Acquittement à distance Effectué. Nombre d'acquittements à distance encore possibles : | Riconoscimento remoto No:
   |  |  |  |  |  *)

(* text list txtLibAp99_3Info (id | default | de | en | fr | it)
  1 | Systemstart |  |  |  | 
   |  |  |  |  |  *)

(* text list txtNoTextList (id | default | de | en | fr | it)
  1 | Keine Textliste gefunden | Keine Textliste gefunden | No text list found | Aucune liste de textes trouvée | Nessun elenco di testi trovato
   |  |  |  |  |  *)
